  rq_init_comm_if_connected(9, "1")
  rq_init_comm_if_connected(2, "2")
  rq_init_comm_if_connected(3, "3")
  rq_init_comm_if_connected(4, "4")
  rq_print_connected_grippers()
  rq_gripper_communication_thread = run rq_gripper_communication()
  set_closed_norm(100.0, 1)
  set_open_norm(0.0, 1)
  set_closed_mm(0.0, 1)
  set_open_mm(50.0, 1)
  set_closed_norm(100.0, 2)
  set_open_norm(0.0, 2)
  set_closed_mm(0.0, 2)
  set_open_mm(50.0, 2)
  set_closed_norm(100.0, 3)
  set_open_norm(0.0, 3)
  set_closed_mm(0.0, 3)
  set_open_mm(50.0, 3)
  set_closed_norm(100.0, 4)
  set_open_norm(0.0, 4)
  set_closed_mm(0.0, 4)
  set_open_mm(50.0, 4)
  rq_current_limit_enabled = False
  while(not rq_gripper_communication_thread_started):
      sleep(0.008)
  end
  # end: URCap Installation Node
  global approach1_p=p[.233098465437, -.416683350523, .053907258737, -2.170613030840, -2.261565526761, -.012256123616]
  global approach1_q=[1.7953318357467651, -1.4227716487697144, 2.1283653418170374, -2.266200681725973, 4.716165542602539, 1.7549076080322266]
  def calculate_point_to_move_towards(feature, direction, position_distance):
    local posDir=[direction[0], direction[1], direction[2]]
    if (norm(posDir) < 1e-6):
      return get_target_waypoint()
    end
    local direction_vector_normalized=normalize(posDir)
    local displacement_pose=p[direction_vector_normalized[0] * position_distance,direction_vector_normalized[1] * position_distance,direction_vector_normalized[2] * position_distance,0,0,0]
    local wanted_displacement_in_base_frame=pose_sub(pose_trans(feature, displacement_pose), feature)
    return pose_add(get_target_waypoint(), wanted_displacement_in_base_frame)
  end
  global approach2_p=p[.356172543172, -.318335465349, .053910905097, -2.170632242458, -2.261543933186, -.012267465714]
  global approach2_q=[2.125020980834961, -1.4233334821513672, 2.1295087973224085, -2.26821293453359, 4.719278335571289, 2.0846056938171387]
  def Pick1():
    $ 13 "Pick1" "noBreak"
    $ 14 "MoveL"
    $ 15 "approach1" "breakAfter"
    movel(approach1_p, a=1.2, v=0.25)
    # begin: URCap Program Node
    #   Source: Robotiq_Grippers, 1.8.6.7016, Robotiq Inc.
    #   Type: Gripper
    $ 16 "Gripper Close (1)"
    if not(gripper_connected[0]):
      popup("Gripper 1 must be connected to run this program.", "No connection", False, True, True)
    end
    if not(rq_is_gripper_activated("1")):
      popup("Gripper 1 is not activated. Go to Installation tab > Gripper to activate it and run the program again.", "Not activated", False, True, True)
    end
    rq_set_pos_spd_for(255, 255, 255, "1")
    rq_wait_pos_spe_for_request(255, 255, 255, "1")
    rq_go_to("1")
    rq_wait("1")
    # end: URCap Program Node
    $ 17 "Direction: Tool Z+"
    global move_thread_flag_17=0
    thread move_thread_17():
      enter_critical
      move_thread_flag_17 = 1
      local towardsPos=calculate_point_to_move_towards(get_forward_kin(), [0.0,0.0,1.0], 0.025)
      movel(towardsPos, a=0.5, v=0.02)
      move_thread_flag_17 = 2
      exit_critical
    end
    move_thread_flag_17 = 0
    move_thread_han_17 = run move_thread_17()
    while (True):
      local targetTcpDirection=get_target_tcp_speed()
      local stepsToRetract=tool_contact(direction=targetTcpDirection)
      if (stepsToRetract > 0):
        kill move_thread_han_17
        stopl(1.0)
        local backTrackMovement=get_actual_joint_positions_history(stepsToRetract)
        local contactPose=get_forward_kin(backTrackMovement)
        local posDir=[targetTcpDirection[0],targetTcpDirection[1],targetTcpDirection[2]]
        local retractTo=contactPose
        if (norm(posDir) > 1e-6):
          local normalizedPosDir=normalize(posDir)
          local additionalRetraction=p[normalizedPosDir[0] * 0.003, normalizedPosDir[1] * 0.003, normalizedPosDir[2] * 0.003, 0, 0, 0]
          retractTo = pose_sub(contactPose, additionalRetraction)
        end
        movel(retractTo, a=1.0, v=0.1)
        $ 18 "Until (tool_contact_detection)"
        # begin: URCap Program Node
        #   Source: Robotiq_Grippers, 1.8.6.7016, Robotiq Inc.
        #   Type: Gripper
        $ 19 "Gripper Move40% (1)"
        if not(gripper_connected[0]):
          popup("Gripper 1 must be connected to run this program.", "No connection", False, True, True)
        end
        if not(rq_is_gripper_activated("1")):
          popup("Gripper 1 is not activated. Go to Installation tab > Gripper to activate it and run the program again.", "Not activated", False, True, True)
        end
        rq_set_pos_spd_for(102, 255, 255, "1")
        rq_wait_pos_spe_for_request(102, 255, 255, "1")
        rq_go_to("1")
        rq_wait("1")
        # end: URCap Program Node
        $ 20 "Direction: Tool Z+"
        global move_thread_flag_20=0
        thread move_thread_20():
          enter_critical
          move_thread_flag_20 = 1
          local towardsPos=calculate_point_to_move_towards(get_forward_kin(), [0.0,0.0,1.0], 0.015)
          movel(towardsPos, a=1.2, v=0.25)
          move_thread_flag_20 = 2
          exit_critical
        end
        move_thread_flag_20 = 0
        move_thread_han_20 = run move_thread_20()
        while (True):
          sleep(1.0E-10)
          if (move_thread_flag_20 > 1):
            join move_thread_han_20
            $ 21 "Until (distance)"
            break
          end
          sync()
        end
        # begin: URCap Program Node
        #   Source: Robotiq_Grippers, 1.8.6.7016, Robotiq Inc.
        #   Type: Gripper
        $ 22 "Gripper Close (1)"
        if not(gripper_connected[0]):
          popup("Gripper 1 must be connected to run this program.", "No connection", False, True, True)
        end
        if not(rq_is_gripper_activated("1")):
          popup("Gripper 1 is not activated. Go to Installation tab > Gripper to activate it and run the program again.", "Not activated", False, True, True)
        end
        rq_set_pos_spd_for(255, 255, 255, "1")
        rq_wait_pos_spe_for_request(255, 255, 255, "1")
        rq_go_to("1")
        rq_wait("1")
        # end: URCap Program Node
        break
      end
      sleep(1.0E-10)
      if (move_thread_flag_17 > 1):
        join move_thread_han_17
        $ 23 "Until (distance)"
        break
      end
      sync()
    end
    $ 24 "approach1" "breakAfter"
    movel(approach1_p, a=1.2, v=0.25)
  end
  def Place2():
    $ 25 "Place2" "noBreak"
    $ 26 "MoveL"
    $ 27 "approach2" "breakAfter"
    movel(approach2_p, a=1.2, v=0.25)
    $ 28 "Direction: Tool Z+"
    global move_thread_flag_28=0
    thread move_thread_28():
      enter_critical
      move_thread_flag_28 = 1
      local towardsPos=calculate_point_to_move_towards(get_forward_kin(), [0.0,0.0,1.0], 1000.0)
      movel(towardsPos, a=0.5, v=0.02)
      move_thread_flag_28 = 2
      exit_critical
    end
    move_thread_flag_28 = 0
    move_thread_han_28 = run move_thread_28()
    while (True):
      local targetTcpDirection=get_target_tcp_speed()
      local stepsToRetract=tool_contact(direction=targetTcpDirection)
      if (stepsToRetract > 0):
        kill move_thread_han_28
        stopl(1.0)
        local backTrackMovement=get_actual_joint_positions_history(stepsToRetract)
        local contactPose=get_forward_kin(backTrackMovement)
        local posDir=[targetTcpDirection[0],targetTcpDirection[1],targetTcpDirection[2]]
        local retractTo=contactPose
        if (norm(posDir) > 1e-6):
          local normalizedPosDir=normalize(posDir)
          local additionalRetraction=p[normalizedPosDir[0] * 0.001, normalizedPosDir[1] * 0.001, normalizedPosDir[2] * 0.001, 0, 0, 0]
          retractTo = pose_sub(contactPose, additionalRetraction)
        end
        movel(retractTo, a=1.0, v=0.1)
        $ 29 "Until (tool_contact_detection)"
        break
      end
      sync()
    end
    # begin: URCap Program Node
    #   Source: Robotiq_Grippers, 1.8.6.7016, Robotiq Inc.
    #   Type: Gripper
    $ 30 "Gripper Move40% (1)"
    if not(gripper_connected[0]):
      popup("Gripper 1 must be connected to run this program.", "No connection", False, True, True)
    end
    if not(rq_is_gripper_activated("1")):
      popup("Gripper 1 is not activated. Go to Installation tab > Gripper to activate it and run the program again.", "Not activated", False, True, True)
    end
    rq_set_pos_spd_for(102, 255, 255, "1")
    rq_wait_pos_spe_for_request(102, 255, 255, "1")
    rq_go_to("1")
    rq_wait("1")
    # end: URCap Program Node
    $ 31 "approach2" "breakAfter"
    movel(approach2_p, a=1.2, v=0.25)
  end
  def Pick2():
    $ 32 "Pick2" "noBreak"
    $ 33 "MoveL"
    $ 34 "approach2" "breakAfter"
    movel(approach2_p, a=1.2, v=0.25)
    # begin: URCap Program Node
    #   Source: Robotiq_Grippers, 1.8.6.7016, Robotiq Inc.
    #   Type: Gripper
    $ 35 "Gripper Close (1)"
    if not(gripper_connected[0]):
      popup("Gripper 1 must be connected to run this program.", "No connection", False, True, True)
    end
    if not(rq_is_gripper_activated("1")):
      popup("Gripper 1 is not activated. Go to Installation tab > Gripper to activate it and run the program again.", "Not activated", False, True, True)
    end
    rq_set_pos_spd_for(255, 255, 255, "1")
    rq_wait_pos_spe_for_request(255, 255, 255, "1")
    rq_go_to("1")
    rq_wait("1")
    # end: URCap Program Node
    $ 36 "Direction: Tool Z+"
    global move_thread_flag_36=0
    thread move_thread_36():
      enter_critical
      move_thread_flag_36 = 1
      local towardsPos=calculate_point_to_move_towards(get_forward_kin(), [0.0,0.0,1.0], 0.025)
      movel(towardsPos, a=0.5, v=0.02)
      move_thread_flag_36 = 2
      exit_critical
    end
    move_thread_flag_36 = 0
    move_thread_han_36 = run move_thread_36()
    while (True):
      local targetTcpDirection=get_target_tcp_speed()
      local stepsToRetract=tool_contact(direction=targetTcpDirection)
      if (stepsToRetract > 0):
        kill move_thread_han_36
        stopl(1.0)
        local backTrackMovement=get_actual_joint_positions_history(stepsToRetract)
        local contactPose=get_forward_kin(backTrackMovement)
        local posDir=[targetTcpDirection[0],targetTcpDirection[1],targetTcpDirection[2]]
        local retractTo=contactPose
        if (norm(posDir) > 1e-6):
          local normalizedPosDir=normalize(posDir)
          local additionalRetraction=p[normalizedPosDir[0] * 0.003, normalizedPosDir[1] * 0.003, normalizedPosDir[2] * 0.003, 0, 0, 0]
          retractTo = pose_sub(contactPose, additionalRetraction)
        end
        movel(retractTo, a=1.0, v=0.1)
        $ 37 "Until (tool_contact_detection)"
        # begin: URCap Program Node
        #   Source: Robotiq_Grippers, 1.8.6.7016, Robotiq Inc.
        #   Type: Gripper
        $ 38 "Gripper Move40% (1)"
        if not(gripper_connected[0]):
          popup("Gripper 1 must be connected to run this program.", "No connection", False, True, True)
        end
        if not(rq_is_gripper_activated("1")):
          popup("Gripper 1 is not activated. Go to Installation tab > Gripper to activate it and run the program again.", "Not activated", False, True, True)
        end
        rq_set_pos_spd_for(102, 255, 255, "1")
        rq_wait_pos_spe_for_request(102, 255, 255, "1")
        rq_go_to("1")
        rq_wait("1")
        # end: URCap Program Node
        $ 39 "Direction: Tool Z+"
        global move_thread_flag_39=0
        thread move_thread_39():
          enter_critical
          move_thread_flag_39 = 1
          local towardsPos=calculate_point_to_move_towards(get_forward_kin(), [0.0,0.0,1.0], 0.015)
          movel(towardsPos, a=1.2, v=0.25)
          move_thread_flag_39 = 2
          exit_critical
        end
        move_thread_flag_39 = 0
        move_thread_han_39 = run move_thread_39()
        while (True):
          sleep(1.0E-10)
          if (move_thread_flag_39 > 1):
            join move_thread_han_39
            $ 40 "Until (distance)"
            break
          end
          sync()
        end
        # begin: URCap Program Node
        #   Source: Robotiq_Grippers, 1.8.6.7016, Robotiq Inc.
        #   Type: Gripper
        $ 41 "Gripper Close (1)"
        if not(gripper_connected[0]):
          popup("Gripper 1 must be connected to run this program.", "No connection", False, True, True)
        end
        if not(rq_is_gripper_activated("1")):
          popup("Gripper 1 is not activated. Go to Installation tab > Gripper to activate it and run the program again.", "Not activated", False, True, True)
        end
        rq_set_pos_spd_for(255, 255, 255, "1")
        rq_wait_pos_spe_for_request(255, 255, 255, "1")
        rq_go_to("1")
        rq_wait("1")
        # end: URCap Program Node
        break
      end
      sleep(1.0E-10)
      if (move_thread_flag_36 > 1):
        join move_thread_han_36
        $ 42 "Until (distance)"
        break
      end
      sync()
    end
    $ 43 "approach2" "breakAfter"
    movel(approach2_p, a=1.2, v=0.25)
  end
  def Place1():
    $ 44 "Place1" "noBreak"
    $ 45 "MoveL"
    $ 46 "approach1" "breakAfter"
    movel(approach1_p, a=1.2, v=0.25)
    $ 47 "Direction: Tool Z+"
    global move_thread_flag_47=0
    thread move_thread_47():
      enter_critical
      move_thread_flag_47 = 1
      local towardsPos=calculate_point_to_move_towards(get_forward_kin(), [0.0,0.0,1.0], 1000.0)
      movel(towardsPos, a=0.5, v=0.02)
      move_thread_flag_47 = 2
      exit_critical
    end
    move_thread_flag_47 = 0
    move_thread_han_47 = run move_thread_47()
    while (True):
      local targetTcpDirection=get_target_tcp_speed()
      local stepsToRetract=tool_contact(direction=targetTcpDirection)
      if (stepsToRetract > 0):
        kill move_thread_han_47
        stopl(1.0)
        local backTrackMovement=get_actual_joint_positions_history(stepsToRetract)
        local contactPose=get_forward_kin(backTrackMovement)
        local posDir=[targetTcpDirection[0],targetTcpDirection[1],targetTcpDirection[2]]
        local retractTo=contactPose
        if (norm(posDir) > 1e-6):
          local normalizedPosDir=normalize(posDir)
          local additionalRetraction=p[normalizedPosDir[0] * 0.001, normalizedPosDir[1] * 0.001, normalizedPosDir[2] * 0.001, 0, 0, 0]
          retractTo = pose_sub(contactPose, additionalRetraction)
        end
        movel(retractTo, a=1.0, v=0.1)
        $ 48 "Until (tool_contact_detection)"
        break
      end
      sync()
    end
    # begin: URCap Program Node
    #   Source: Robotiq_Grippers, 1.8.6.7016, Robotiq Inc.
    #   Type: Gripper
    $ 49 "Gripper Move40% (1)"
    if not(gripper_connected[0]):
      popup("Gripper 1 must be connected to run this program.", "No connection", False, True, True)
    end
    if not(rq_is_gripper_activated("1")):
      popup("Gripper 1 is not activated. Go to Installation tab > Gripper to activate it and run the program again.", "Not activated", False, True, True)
    end
    rq_set_pos_spd_for(102, 255, 255, "1")
    rq_wait_pos_spe_for_request(102, 255, 255, "1")
    rq_go_to("1")
    rq_wait("1")
    # end: URCap Program Node
    $ 50 "approach1" "breakAfter"
    movel(approach1_p, a=1.2, v=0.25)
  end
  $ 2 "BeforeStart"
  # begin: URCap Program Node
  #   Source: Robotiq_Grippers, 1.8.6.7016, Robotiq Inc.
  #   Type: Gripper Activate
  $ 3 "Gripper Activate"

  kill rq_gripper_communication_thread
  rq_gripper_communication_thread_started = False
  rq_close_gripper_socket("1")
  rq_close_gripper_socket("2")
  rq_close_gripper_socket("3")
  rq_close_gripper_socket("4")

  rq_init_comm_if_connected(9, "1")
  rq_init_comm_if_connected(2, "2")
  rq_init_comm_if_connected(3, "3")
  rq_init_comm_if_connected(4, "4")
  rq_print_connected_grippers()
  rq_gripper_communication_thread = run rq_gripper_communication()

  while(not rq_gripper_communication_thread_started):
      sleep(0.008)
  end

  rq_set_max_current_for_all_grippers()

  reset_and_activate = False

  rq_activate_all_grippers(False)
  # end: URCap Program Node
  while (True):
    $ 4 "Robot Program"
    $ 5 "Call Pick1"
    Pick1()
    # begin: URCap Program Node
    #   Source: Robotiq_Grippers, 1.8.6.7016, Robotiq Inc.
    #   Type: Grip Check
    $ 6 "Grip Check"
    # begin: URCap Program Node
    #   Source: Robotiq_Grippers, 1.8.6.7016, Robotiq Inc.
    #   Type: If
    $ 7 "If object detected          " "noBreak"
    if (rq_is_object_detected(1)):
      $ 8 "Call Place2" "noBreak"
      Place2()
      # end: URCap Program Node
    end
    # end: URCap Program Node
    $ 9 "Call Pick2"
    Pick2()
    # begin: URCap Program Node
    #   Source: Robotiq_Grippers, 1.8.6.7016, Robotiq Inc.
    #   Type: Grip Check
    $ 10 "Grip Check"
    # begin: URCap Program Node
    #   Source: Robotiq_Grippers, 1.8.6.7016, Robotiq Inc.
    #   Type: If
    $ 11 "If object detected          " "noBreak"
    if (rq_is_object_detected(1)):
      $ 12 "Call Place1" "noBreak"
      Place1()
      # end: URCap Program Node
    end
    # end: URCap Program Node
  end
end
